FUNCTION_BLOCK FB_Station IMPLEMENTS IStation
VAR_INPUT
END_VAR
VAR_OUTPUT
END_VAR
VAR
END_VAR

END_FUNCTION_BLOCK

(* stored: Version 1.1.0.1, ProductVersion 3.1.4024.6
   POU FB_Station: Id {f7551307-30e4-45a3-8d86-064d6f4dc85f}, SpecialFunc None *)
